(* CODESYS project EtherCat-demo-projectSoE.project
   Description: This example shows how to read and write IDN’s with ServoDrive over EtherCAT. As hardware a Rexroth IndraDrive is used (the exact specification can be found under the point “Additional Requirements”). It is also possible to switch to device to another one which can ServoDrive over EtherCAT.
   Title: EtherCAT SoE

Project tree, tasks and I/O mapping:
  Device : CODESYS Control RTE V3 x64, CODESYS, version 3.5.21.30
    application Application
      libraries: Standard, * (System); CAA Types Extern, 3.5.17.0 (CAA Technical Workgroup); SM3_Basic, 4.19.0.0 (CODESYS); SM3_Basic_Visu, 4.19.0.0 (CODESYS); SM3_CamBuilder, 4.19.0.0 (CODESYS); SM3_Shared, * (CODESYS); SM3_StringUtils, 4.19.0.0 (CODESYS); SM3_TrajectoryGeneration, 4.18.0.0 (CODESYS); SM3_Transformation, 4.19.0.0 (CODESYS)
      task MainTask (cyclic, interval t#20ms, priority 1) calls SoE
      task EtherCAT_Task (cyclic, interval t#4ms, priority 0) calls EtherCAT_Master.EtherCAT_Task
      program SoE [ST]
      license
      program POU [CFC]
    EtherCAT_Master : EtherCAT Master, CODESYS, version 4.9.0.0 (disabled)
        settings: NetworkName = '\Device\NPF_{C7E8FB72-3D27-40B3-9AF5-4A504186529A}'; SrcAddress1 = 10; SrcAddress2 = 3441249734
      IndraDrive_Basic_Cs : IndraDrive Basic Cs, BoschRexroth, version Revision=16#00000001
          settings: DC sync0 cycletime = 4000; DC enable = 1; DC sync0 factor = 'x 1'; DC sync0 shift time = 500; DC sync1 cycletime = 4000; DC sync1 enable = 1; DC sync1 factor = ''; DC sync1 shift time = 0; DCSetting = 0
          unmapped channels: Master control word, Position command value, Drive status word, Position feedback value 1
    EtherCAT_Master_SoftMotion : EtherCAT Master SoftMotion, CODESYS, version 4.10.0.0
        settings: NetworkName = 'Ethernet 5'; NetworkName = "Ethernet 5"; SrcAddress1 = 22599; SrcAddress2 = 3396740476
      A6N_Servo_Driver : A6N_sAxis_V0.02, STEPPERONLINE, order no. A6N Servo Driver, version Revision=16#00002EF8
          settings: DC sync0 cycletime = 4000; DC sync1 cycletime = 4000
          unmapped channels: Controlword, Target position, Touch probe function, Physical outputs, Error code, Statusword, Position actual value, Torque actual value, Following error actual value, Touch probe status, Touch probe pos1 pos value, Touch probe pos2 pos value, Digital inputs
      A6N_Servo_Driver_1 : A6N_sAxis_V0.02, STEPPERONLINE, order no. A6N Servo Driver, version Revision=16#00002EF8
          settings: DC sync0 cycletime = 4000; DC sync1 cycletime = 4000
          unmapped channels: Controlword, Target position, Touch probe function, Physical outputs, Error code, Statusword, Position actual value, Torque actual value, Following error actual value, Touch probe status, Touch probe pos1 pos value, Touch probe pos2 pos value, Digital inputs
        Axis1 : SM_Drive_GenericDSP402, CODESYS, order no. 0, version 4.19.0.0
            settings: wDriveID = 0; AdrOffset_8010 = 0; BitOffset_8010 = 0; BitLength_8010 = 16; Address_8010 = '%QW0'; Type_8010 = 'UINT'; AddressPointer_8010 = ADR(%QW0); AdrOffset_8020 = 4; BitOffset_8020 = 0; BitLength_8020 = 32; Address_8020 = '%QD1'; Type_8020 = 'DINT'; AddressPointer_8020 = ADR(%QD1); AdrOffset_8030 = 4294967295; BitOffset_8030 = 0; BitLength_8030 = 0; Address_8030 = ''; Type_8030 = ''; AddressPointer_8030 = 0; AdrOffset_8040 = 4294967295; BitOffset_8040 = 0; BitLength_8040 = 0; Address_8040 = ''; Type_8040 = ''; AddressPointer_8040 = 0; AdrOffset_8050 = 4294967295; BitOffset_8050 = 0; BitLength_8050 = 0; Address_8050 = ''; Type_8050 = ''; AddressPointer_8050 = 0; AdrOffset_8060 = 8; BitOffset_8060 = 0; BitLength_8060 = 16; Address_8060 = '%QW4'; Type_8060 = 'UINT'; AddressPointer_8060 = ADR(%QW4); AdrOffset_8070 = 4294967295; BitOffset_8070 = 0; BitLength_8070 = 0;
              Address_8070 = ''; Type_8070 = ''; AddressPointer_8070 = 0; AdrOffset_8080 = 4294967295; BitOffset_8080 = 0; BitLength_8080 = 0; Address_8080 = ''; Type_8080 = ''; AddressPointer_8080 = 0; AdrOffset_8090 = 12; BitOffset_8090 = 0; BitLength_8090 = 32; Address_8090 = '%QD3'; Type_8090 = 'UDINT'; AddressPointer_8090 = ADR(%QD3); AdrOffset_8510 = 2; BitOffset_8510 = 0; BitLength_8510 = 16; Address_8510 = '%IW1'; Type_8510 = 'UINT'; AddressPointer_8510 = ADR(%IW1); AdrOffset_8520 = 4; BitOffset_8520 = 0; BitLength_8520 = 32; Address_8520 = '%ID1'; Type_8520 = 'DINT'; AddressPointer_8520 = ADR(%ID1); AdrOffset_8530 = 4294967295; BitOffset_8530 = 0; BitLength_8530 = 0; Address_8530 = ''; Type_8530 = ''; AddressPointer_8530 = 0; AdrOffset_8540 = 8; BitOffset_8540 = 0; BitLength_8540 = 16; Address_8540 = '%IW4'; Type_8540 = 'INT'; AddressPointer_8540 = ADR(%IW4); AdrOffset_8550 = 4294967295;
              BitOffset_8550 = 0; BitLength_8550 = 0; Address_8550 = ''; Type_8550 = ''; AddressPointer_8550 = 0; AdrOffset_8560 = 28; BitOffset_8560 = 0; BitLength_8560 = 32; Address_8560 = '%ID7'; Type_8560 = 'UDINT'; AddressPointer_8560 = ADR(%ID7); AdrOffset_8570 = 16; BitOffset_8570 = 0; BitLength_8570 = 16; Address_8570 = '%IW8'; Type_8570 = 'UINT'; AddressPointer_8570 = ADR(%IW8); AdrOffset_8580 = 20; BitOffset_8580 = 0; BitLength_8580 = 32; Address_8580 = '%ID5'; Type_8580 = 'DINT'; AddressPointer_8580 = ADR(%ID5); AdrOffset_8590 = 4294967295; BitOffset_8590 = 0; BitLength_8590 = 0; Address_8590 = ''; Type_8590 = ''; AddressPointer_8590 = 0; AdrOffset_8600 = 24; BitOffset_8600 = 0; BitLength_8600 = 32; Address_8600 = '%ID6'; Type_8600 = 'DINT'; AddressPointer_8600 = ADR(%ID6); AdrOffset_8600 = 4294967295; BitOffset_8600 = 0; BitLength_8600 = 0; Address_8610 = ''; Type_8610 = '';
              AddressPointer_8610 = 0; AdrOffset_8620 = 12; BitOffset_8620 = 0; BitLength_8620 = 32; Address_8620 = '%ID3'; Type_8620 = 'DINT'; AddressPointer_8620 = ADR(%ID3)
    SoftMotion General Axis Pool : SoftMotion General Axis Pool, CODESYS, version 4.11.0.0
  00000000-0000-0000-0000-000000000000|C:\Users\m.lamp\Documents\license.txt
*)

// Device/Application/SoE
PROGRAM SoE
VAR
	iState			: INT; (* state variable *)
	
	Read			: ETC_SoE_IDNRead; (* Instance to read an IDN. *)
	Read4			: ETC_SoE_IDNRead4; (* Instance to read an IDN with a maximum of 4 bytes. *)
	Write			: ETC_SoE_IDNWrite; (* Instance to write an IDN. *)
	Write4			: ETC_SoE_IDNWrite4; (* Instance to write an IDN with a maximum of 4 bytes. *)
	Command			: ETC_SoE_Cmd;
	
	udiRead			: UDINT; (* The read value of the IDN. *)
	uiWrite			: UINT; (* The value to be written to the IDN. *)
	uiReadWritten	: UINT; (* The read value of the IDN, written in the step before. *)
	
	abyRead			: ARRAY[1..4] OF BYTE; (* Read EtherCAT IDN value *)
	abyWrite		: ARRAY[1..4] OF BYTE := [8, 9, 0, 0]; (* Write a value with a maximum of 4 bytes. *)
END_VAR

(* Global instance of the IoDrvEtherCAT function block.*)
EtherCAT_Master_SoftMotion();

CASE iState OF
	0:
		(* Wait for the EtherCAT to be ready. *)
		IF Ethercat_Master.xConfigFinished THEN
			iState := iState + 1;
		END_IF
		
	1: (* Read the IDN with the number 32. The value at byElem indicates that the value of the IDN is written. Other numbers are 
		  possible. Have a look at the "IODrvEtherCAT" lib under "ServoDrive_o_Ethercat".  The device address is 1001 (Look at the device
		  under the "Slave" tab).usiCom = 1, because the first master is used. A buffer is set, to where the value will be written*)
		Read(xExecute := TRUE, usiCom := 1, uiDevice := 1001, wIDN := 32, byElem := 7, udiTimeOut := 1000, pBuffer := ADR(udiRead), szSize := SIZEOF(udiRead));
		
		(* When the value is read without an error, go to the next step. *)
		IF Read.xDone THEN
			iState := iState + 1;
			Read(xExecute := FALSE);
		ELSIF Read.xError THEN
			iState := 32767;
		END_IF	
		
	2: (* Write a IDN with number 33 and the value 11 at the same device. *)
		uiWrite := 11;
		Write(xExecute := TRUE, usiCom := 1, uiDevice := 1001, wIDN := 33, byElem := 7, pBuffer := ADR(uiWrite), szSize := SIZEOF(uiWrite), udiTimeOut := 1000);
		
		(* When the value is written without an error, go TO the next step. *)
		IF Write.xDone THEN
			iState := iState + 1;
			Write(xExecute := FALSE);
		ELSIF Write.xError THEN
			iState := 32767;
		END_IF
		
	3: (* Read the IDN number 33, which was written in the step before. *)
		Read(xExecute := TRUE, usiCom := 1, uiDevice := 1001, wIDN := 33, byElem := 7, pBuffer := ADR(uiReadWritten), szSize := SIZEOF(uiReadWritten), udiTimeOut := 1000);
		
		IF Read.xDone THEN
			iState := iState + 1;
			Read(xExecute := FALSE);
		ELSIF Read.xError THEN
			iState := 32767;
		END_IF	
		
	4: (* Write a IDN with number 34 from an array to the device. *)
		Write4(xExecute := TRUE, usiCom := 1, uiDevice := 1001, wIDN := 34, byElem := 7, abyData := abyWrite, usiDataLength := 2, udiTimeOut := 1000);
		
		IF Write4.xDone THEN
			iState := iState + 1;
			Write4(xExecute := FALSE);
		ELSIF Write4.xError THEN
			iState := 32767;
		END_IF
		
	5: (* Read the IDN number 34, which was written in the step before. *)
		Read4(xExecute := TRUE, usiCom := 1, uiDevice := 1001, wIDN := 34, byElem := 7, udiTimeOut := 1000);
		
		IF Read4.xDone THEN
			abyRead := Read4.abyData;	
			iState := iState + 1;
			Read4(xExecute := FALSE);
		ELSIF Read4.xError THEN
			iState := 32767;
		END_IF

	32767: (* error *) ;	
	
END_CASE

END_PROGRAM

// Device/Application/POU
PROGRAM POU
VAR
END_VAR

END_PROGRAM
